PROGRAM DiagnosticEtherCAT
VAR
END_VAR
(* End *)

(* Diagnosis of the EtherCat System *)

	fbDiagnosticEtherCAT(bEnable :=	TRUE);
	
(* End *)

END_PROGRAM

(* stored: Version 1.1.0.1, ProductVersion 3.1.4018.5
   POU DiagnosticEtherCAT: Id {82c1e4ad-6a0e-4cd2-96b4-e5f30f640e81}, SpecialFunc None *)
